TYPE
    ST_Manual_Allocate :
    STRUCT
        WorkZone_Press      : ST_SignleValve;
        WorkZone_Plug       : ST_SignleValve; //定位銷
        ChargeZone_Plug     : ST_SignleValve; //定位銷
        TransmitCVZone_Plug : ST_SignleValve; //定位銷
        Axis                : ST_Manual_Axis; // RoundBelt Axis controll
		
    END_STRUCT
END_TYPE

(* stored: Version 1.1.0.1, ProductVersion 3.1.4024.13
   DUT ST_Manual_Allocate: Id {f49b177b-3e6b-4723-93fa-1918947532c6} *)
